TYPE Mat34 : ARRAY[1..3, 1..4] OF LREAL; END_TYPE

(* stored: Version 1.1.0.1, ProductVersion 3.1.4024.12
   DUT Mat34: Id {720198b6-e5dc-4e97-aa09-45ca28de840d} *)
